// TIA Portal V20 export
DATA_BLOCK "Tempering_HMI"   // DB107
AUTHOR : Siemens AG
FAMILY : ServiceControl
VERSION : 4.0
// stored: InstanceOfName ServiceParameterHMITempering, InstanceOfType FB
"ServiceParameterHMITempering"
   // VAR_INPUT
   //    Id { ExternalAccessible := 'False'; ExternalVisible := 'False'; ExternalWritable := 'False'} : USInt;
   //    Setup { ExternalAccessible := 'False'; ExternalVisible := 'False'; ExternalWritable := 'False'} : DB_ANY;
   //    ProcedureCur { ExternalAccessible := 'False'; ExternalVisible := 'False'; ExternalWritable := 'False'} : DWord;
   //    ProcedureReq { ExternalAccessible := 'False'; ExternalVisible := 'False'; ExternalWritable := 'False'} : DWord;
   // END_VAR
   // VAR_IN_OUT
   //    ConfigurationParameterAnalog : Array[*] of "UDT_MTP_AnaServParam";
   //    ConfigurationParameterDigital : Array[*] of "UDT_MTP_DIntServParam";
   //    ConfigurationParameterBinary : Array[*] of "UDT_MTP_BinServParam";
   //    ConfigurationParameterString : Array[*] of "UDT_MTP_StringServParam";
   //    ProcedureParameterAnalog : Array[*] of "UDT_MTP_AnaServParam";
   //    ProcedureParameterDigital : Array[*] of "UDT_MTP_DIntServParam";
   //    ProcedureParameterBinary : Array[*] of "UDT_MTP_BinServParam";
   //    ProcedureParameterString : Array[*] of "UDT_MTP_StringServParam";
   //    ProcessValueInAnalog : Array[*] of "UDT_MTP_AnaProcessValueIn";
   //    ProcessValueInDigital : Array[*] of "UDT_MTP_DIntProcessValueIn";
   //    ProcessValueInBinary : Array[*] of "UDT_MTP_BinProcessValueIn";
   //    ProcessValueInString : Array[*] of "UDT_MTP_StringProcessValueIn";
   //    ProcessValueOutAnalog : Array[*] of "UDT_MTP_AnaProcessValueOut";
   //    ProcessValueOutDigital : Array[*] of "UDT_MTP_DIntProcessValueOut";
   //    ProcessValueOutBinary : Array[*] of "UDT_MTP_BinProcessValueOut";
   //    ProcessValueOutString : Array[*] of "UDT_MTP_StringProcessValueOut";
   //    ReportValueAnalog : Array[*] of "UDT_MTP_AnaReportValue";
   //    ReportValueDigital : Array[*] of "UDT_MTP_DIntReportValue";
   //    ReportValueBinary : Array[*] of "UDT_MTP_BinReportValue";
   //    ReportValueString : Array[*] of "UDT_MTP_StringReportValue";
   // END_VAR
   // VAR
   //    statTotalConfigParameters { ExternalAccessible := 'False'; ExternalVisible := 'False'; ExternalWritable := 'False'} : Int;
   //    statTotalProcedureParameters { ExternalAccessible := 'False'; ExternalVisible := 'False'; ExternalWritable := 'False'} : Int;
   //    statTotalProcessInValues { ExternalAccessible := 'False'; ExternalVisible := 'False'; ExternalWritable := 'False'} : Int;
   //    statTotalProcessOutValues { ExternalAccessible := 'False'; ExternalVisible := 'False'; ExternalWritable := 'False'} : Int;
   //    statTotalReportValues { ExternalAccessible := 'False'; ExternalVisible := 'False'; ExternalWritable := 'False'} : Int;
   //    StatConfigAnalog { ExternalAccessible := 'False'; ExternalVisible := 'False'; ExternalWritable := 'False'} : Array[0..0] of "UDT_Service_AnaServParam";
   //    StatConfigDigital { ExternalAccessible := 'False'; ExternalVisible := 'False'; ExternalWritable := 'False'} : Array[0..0] of "UDT_Service_DintServParam";
   //    StatConfigBinary { ExternalAccessible := 'False'; ExternalVisible := 'False'; ExternalWritable := 'False'} : Array[0..0] of "UDT_Service_BinServParam";
   //    StatConfigString { ExternalAccessible := 'False'; ExternalVisible := 'False'; ExternalWritable := 'False'} : Array[0..0] of "UDT_Service_StringServParam";
   //    StatProcedureAnalog { ExternalAccessible := 'False'; ExternalVisible := 'False'; ExternalWritable := 'False'} : Array[0..2] of "UDT_Service_AnaServParam";
   //    StatProcedureDigital { ExternalAccessible := 'False'; ExternalVisible := 'False'; ExternalWritable := 'False'} : Array[0..0] of "UDT_Service_DintServParam";
   //    StatProcedureBinary { ExternalAccessible := 'False'; ExternalVisible := 'False'; ExternalWritable := 'False'} : Array[0..0] of "UDT_Service_BinServParam";
   //    StatProcedureString { ExternalAccessible := 'False'; ExternalVisible := 'False'; ExternalWritable := 'False'} : Array[0..0] of "UDT_Service_StringServParam";
   //    stat16ProceReqIndex { ExternalAccessible := 'False'; ExternalVisible := 'False'; ExternalWritable := 'False'} : Int;
   //    stat16ProceCurIndex { ExternalAccessible := 'False'; ExternalVisible := 'False'; ExternalWritable := 'False'} : Int;
   //    stat16ProcParaStartIndex { ExternalAccessible := 'False'; ExternalVisible := 'False'; ExternalWritable := 'False'} : Int;
   //    stat16ProcParaEndIndex { ExternalAccessible := 'False'; ExternalVisible := 'False'; ExternalWritable := 'False'} : Int;
   //    stat32PrecedureProcessOutMap { ExternalAccessible := 'False'; ExternalVisible := 'False'; ExternalWritable := 'False'} : DWord;
   //    stat32PrecedureProcessInMap { ExternalAccessible := 'False'; ExternalVisible := 'False'; ExternalWritable := 'False'} : DWord;
   //    stat32PrecedureReportMap { ExternalAccessible := 'False'; ExternalVisible := 'False'; ExternalWritable := 'False'} : DWord;
   //    ConfigParaType : "UDT_Service_ConfigParaIndexType";
   //    ProcedureParaType : "UDT_Service_ProceParaValueIndexType";
   //    ProcessInValueType : "UDT_Service_ProceParaValueIndexType";
   //    ProcessOutValueType : "UDT_Service_ProceParaValueIndexType";
   //    ReportValueType : "UDT_Service_ProceParaValueIndexType";
   //    ConfigAna : Array[0..0] of "UDT_MTP_AnaServParam";
   //    ConfigDint : Array[0..0] of "UDT_MTP_DIntServParam";
   //    ConfigBin : Array[0..0] of "UDT_MTP_BinServParam";
   //    ConfigString : Array[0..0] of "UDT_MTP_StringServParam";
   //    ProcedureAna : Array[0..2] of "UDT_MTP_AnaServParam";
   //    ProcedureDint : Array[0..0] of "UDT_MTP_DIntServParam";
   //    ProcedureBin : Array[0..0] of "UDT_MTP_BinServParam";
   //    ProcedureString : Array[0..0] of "UDT_MTP_StringServParam";
   //    ProcessInAna : Array[0..0] of "UDT_MTP_AnaProcessValueIn";
   //    ProcessInDint : Array[0..0] of "UDT_MTP_DIntProcessValueIn";
   //    ProcessInBin : Array[0..0] of "UDT_MTP_BinProcessValueIn";
   //    ProcessInString : Array[0..0] of "UDT_MTP_StringProcessValueIn";
   //    ProcessOutAna : Array[0..2] of "UDT_MTP_AnaProcessValueOut";
   //    ProcessOutDint : Array[0..0] of "UDT_MTP_DIntProcessValueOut";
   //    ProcessOutBin : Array[0..0] of "UDT_MTP_BinProcessValueOut";
   //    ProcessOutString : Array[0..0] of "UDT_MTP_StringProcessValueOut";
   //    ReportAna : Array[0..2] of "UDT_MTP_AnaReportValue";
   //    ReportDint : Array[0..0] of "UDT_MTP_DIntReportValue";
   //    ReportBin : Array[0..0] of "UDT_MTP_BinReportValue";
   //    ReportString : Array[0..0] of "UDT_MTP_StringReportValue";
   //    statInternalCurProcParameter { ExternalAccessible := 'False'; ExternalVisible := 'False'; ExternalWritable := 'False'} : Array[0..31] of "UDT_Service_Parameter";
   //    statLasProcedureCur { ExternalAccessible := 'False'; ExternalVisible := 'False'; ExternalWritable := 'False'} : DWord;
   //    statLasProcedureReq { ExternalAccessible := 'False'; ExternalVisible := 'False'; ExternalWritable := 'False'} : DWord;
   //    statLastReqProcedSelected { ExternalAccessible := 'False'; ExternalVisible := 'False'; ExternalWritable := 'False'} : Bool;
   //    StatLastProceselReport { ExternalAccessible := 'False'; ExternalVisible := 'False'; ExternalWritable := 'False'} : Bool;
   //    StatLastProceselProcessOut { ExternalAccessible := 'False'; ExternalVisible := 'False'; ExternalWritable := 'False'} : Bool;
   //    StatLastProceselProcessIn { ExternalAccessible := 'False'; ExternalVisible := 'False'; ExternalWritable := 'False'} : Bool;
   // END_VAR
BEGIN
END_DATA_BLOCK
